ABB RobotStudio station: Practica1.rspag

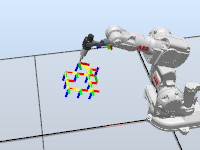
--- station ---
Station Practica1 (saved by RobotStudio 20.4.9280.0)
Controller Controlador2
  mechanical unit ROB_1: IRB140_6_81_C_03, 6 joints, base frame (0, 0, 0) mm
Layout (positions relative to the parent item):
  - IRB140_6_81_C_03 [mechanism, from Robots\IRB140_6_81_C_G_03.rslib] at (0, 0, 0) mm; joint values [0, 0.0792, -0.4687, 0, 0.9131, 0] (rad or m)
  - MyTool [mechanism, from Training Objects\myTool.rslib] at (506.29, 0, 822.68) mm, rotated rx -180 ry 60 rz -180 deg
Attachment: MyTool is attached to IRB140_6_81_C_03 / Link6

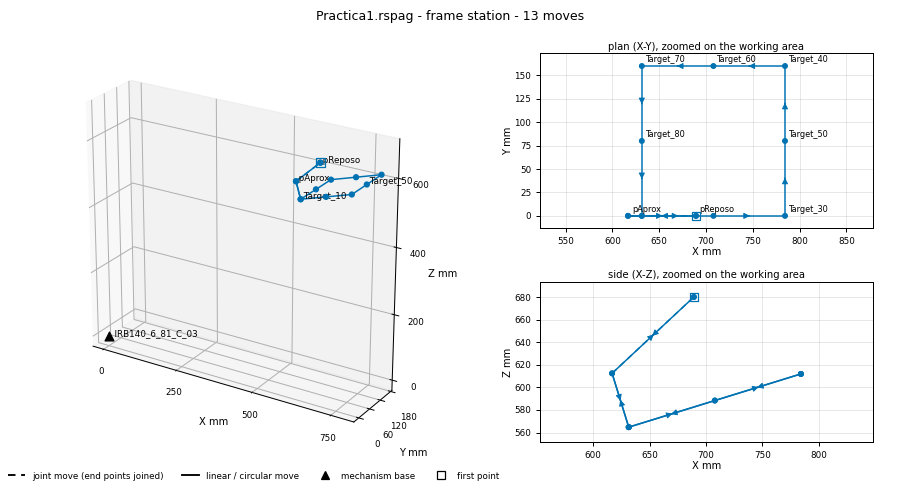
[picture p0: tool path of Practica1.rspag in frame station, 13 of 13 moves have a stored position in this frame; points joined in program order, loops and branches not executed]
--- Backups/Controlador2/RAPID/TASK1/PROGMOD/CalibData.mod ---
MODULE CalibData
    PERS tooldata MyTool:=[TRUE,[[31.792631019,0,229.638935148],[0.945518576,0,0.325568154,0]],[1,[0,0,1],[1,0,0,0],0,0,0]];
    TASK PERS wobjdata Workobject_1:=[FALSE,TRUE,"",[[583.696957106,0,550],[0.988787178,0,-0.149331565,0]],[[0,0,0],[1,0,0,0]]];
ENDMODULE

--- Backups/Controlador2/RAPID/TASK1/PROGMOD/Module1.mod ---
MODULE Module1
        CONST robtarget pReposo:=[[689.268558126,0,680.330541406],[0.19080893,0,0.981627196,0],[0,0,0,0],[9E+09,9E+09,9E+09,9E+09,9E+09,9E+09]];
    CONST robtarget pAprox:=[[50.000102701,0,50.026858914],[-0.000000223,0,1,0],[-1,0,-1,0],[9E+09,9E+09,9E+09,9E+09,9E+09,9E+09]];
    CONST robtarget Target_10:=[[50,0,0],[0,0,1,0],[0,0,-1,0],[9E+09,9E+09,9E+09,9E+09,9E+09,9E+09]];
    CONST robtarget Target_20:=[[130,0,0],[0,0,1,0],[-1,0,-1,0],[9E+09,9E+09,9E+09,9E+09,9E+09,9E+09]];
    CONST robtarget Target_30:=[[210,0,0],[0,0,1,0],[-1,0,-1,0],[9E+09,9E+09,9E+09,9E+09,9E+09,9E+09]];
    CONST robtarget Target_50:=[[210,80,0],[0,0,1,0],[0,-1,0,0],[9E+09,9E+09,9E+09,9E+09,9E+09,9E+09]];
    CONST robtarget Target_40:=[[210,160,0],[0,0,1,0],[0,-1,0,0],[9E+09,9E+09,9E+09,9E+09,9E+09,9E+09]];
    CONST robtarget Target_60:=[[130,160,0],[0,0,1,0],[0,-1,0,0],[9E+09,9E+09,9E+09,9E+09,9E+09,9E+09]];
    CONST robtarget Target_70:=[[50,160,0],[0,0,1,0],[0,-1,0,0],[9E+09,9E+09,9E+09,9E+09,9E+09,9E+09]];
    CONST robtarget Target_80:=[[50,80,0],[0,0,1,0],[0,-1,0,0],[9E+09,9E+09,9E+09,9E+09,9E+09,9E+09]];
!***********************************************************
    !
    ! Módulo:  Module1
    !
    ! Descripción:
    !   <Introduzca la descripción aquí>
    !
    ! Autor: franc
    !
    ! Versión: 1.0
    !
    !***********************************************************


    !***********************************************************
    !
    ! Procedimiento Main
    !
    !   Este es el punto de entrada de su programa
    !
    !***********************************************************
    PROC main()
        !Añada aquí su código
        Path_10;
    ENDPROC
    PROC Path_10()
        MoveJ pReposo,v100,z100,MyTool\WObj:=wobj0;
        MoveL pAprox,v100,z100,MyTool\WObj:=Workobject_1;
        MoveL Target_10,v100,fine,MyTool\WObj:=Workobject_1;
        MoveL Target_20,v100,fine,MyTool\WObj:=Workobject_1;
        MoveL Target_30,v100,fine,MyTool\WObj:=Workobject_1;
        MoveL Target_50,v100,fine,MyTool\WObj:=Workobject_1;
        MoveL Target_40,v100,fine,MyTool\WObj:=Workobject_1;
        MoveL Target_60,v100,fine,MyTool\WObj:=Workobject_1;
        MoveL Target_70,v100,fine,MyTool\WObj:=Workobject_1;
        MoveL Target_80,v100,fine,MyTool\WObj:=Workobject_1;
        MoveL Target_10,v100,fine,MyTool\WObj:=Workobject_1;
        MoveL pAprox,v100,z100,MyTool\WObj:=Workobject_1;
        MoveJ pReposo,v100,fine,MyTool\WObj:=wobj0;
    ENDPROC
ENDMODULE
